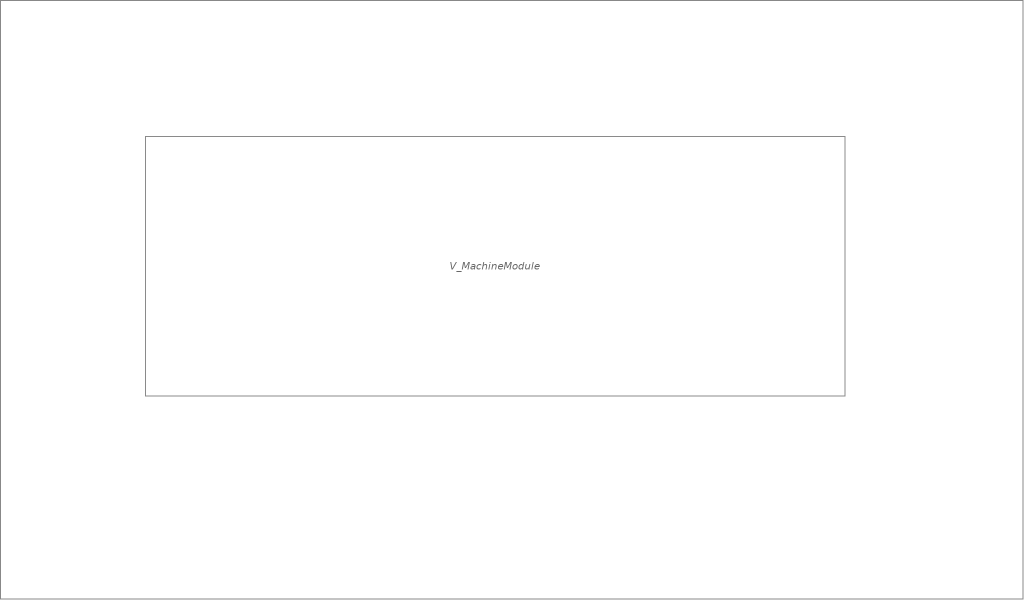
VISUALIZATION V_Main  // 1024x600
    Frame (145,136 700x260)
        shows V_MachineModule(HMI := MAIN.Seedra.PackMLBaseModule_HMI)
END_VISUALIZATION

(* stored: Version 1.1.0.1, ProductVersion 3.1.4024.15
   Visu V_Main: Id {a605f27f-6b24-0012-2ed8-5e678528cd71} *)
